// TIA Portal V17 export
// export: Created 2025-04-09T07:53:26.3404898Z, ExportSetting WithDefaults, DisplayName Totally Integrated Automation Portal, DisplayVersion V17, DisplayName TIA Portal Openness, DisplayVersion V17, DisplayName TIA Portal Version Control Interface, DisplayVersion V17, DisplayName STEP 7 Professional, DisplayVersion V17, DisplayName STEP 7 Safety, DisplayVersion V17, DisplayName WinCC Advanced, DisplayVersion V17
VAR_GLOBAL   // PLC tag table "Input"
   I0 AT %I22.0 : Bool;
   I1 AT %I22.1 : Bool;
   I2 AT %I22.2 : Bool;
   I3 AT %I22.3 : Bool;
   I4 AT %I22.4 : Bool;
   I5 AT %I22.5 : Bool;
   I6 AT %I22.6 : Bool;
   I7 AT %I22.7 : Bool;
   I8 AT %I23.0 : Bool;
   I9 AT %I23.1 : Bool;
   I10 AT %I23.2 : Bool;
   I11 AT %I23.3 : Bool;
END_VAR
